// TIA Portal V19 export
FUNCTION_BLOCK "Convoyer7"   // FB6, F_LAD
{ S7_Optimized_Access := 'TRUE' }
   VAR_INPUT
      InverterStatus : "LDrvSafe_typeSinaTlg30Status";
      ESTOP : Bool;
      LIGHT_CURTAIN : Bool;
      PROCES_STAMPING : Bool;
      DOOR : Bool;
      FRQ_FEEDBACK : Bool;
      RESET : Bool;
   END_VAR
   VAR_OUTPUT
      InverterControl : "LDrvSafe_typeSinaTlg30Control";
      SAFETY_OK : Bool;
      INVERTER_OK : Bool;
      FRQ_NOK : Bool;
      REQ_RESET_ESTOP : Bool;
      SAFETY_VALVE : Bool;
   END_VAR
   VAR
      ESTOP_ON : Bool;
      INVERTER_FAULT : Bool;
      ESTOP1_Instance : ESTOP1;
      LDrvSafe_SinaTlg30Control_Instance : "LDrvSafe_SinaTlg30Control";
      LDrvSafe_SinaTlg30Status_Instance : "LDrvSafe_SinaTlg30Status";
   END_VAR
BEGIN

REGION Network 1
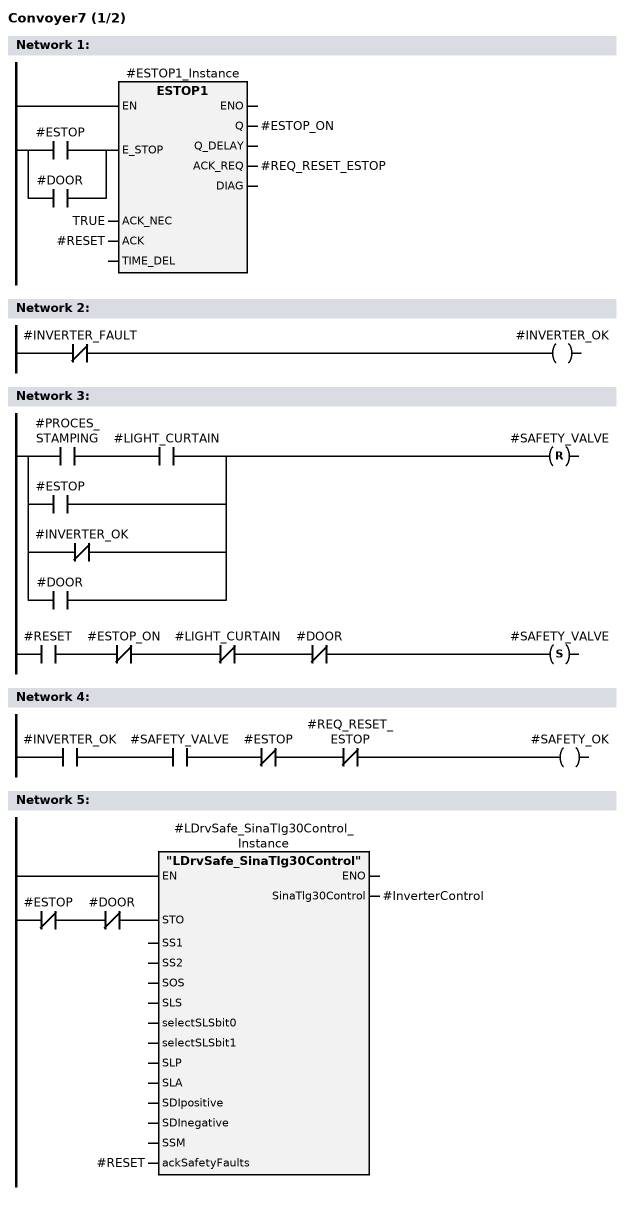
   RUNG wire#powerrail
      #ESTOP1_Instance.ESTOP1(E_STOP := wire#w1, ACK_NEC := TRUE, ACK := #RESET, TIME_DEL :=, Q => #ESTOP_ON, Q_DELAY =>, ACK_REQ => #REQ_RESET_ESTOP, DIAG =>)
   END_RUNG
   RUNG wire#powerrail
      Contact( #ESTOP )
   END_RUNG wire#w1
   RUNG wire#powerrail
      Contact( #DOOR )
   END_RUNG wire#w1
   // the same network as SCL:
   #ESTOP1_Instance(E_STOP := #ESTOP OR #DOOR,   // ESTOP1
                    ACK_NEC := TRUE,
                    ACK := #RESET,
                    Q => #ESTOP_ON,
                    ACK_REQ => #REQ_RESET_ESTOP);
END_REGION

REGION Network 2
   RUNG wire#powerrail
      I_Contact( #INVERTER_FAULT )
      Coil( #INVERTER_OK )
   END_RUNG
   // the same network as SCL:
   #INVERTER_OK := NOT #INVERTER_FAULT;
END_REGION

REGION Network 3
   RUNG wire#powerrail
      Contact( #PROCES_STAMPING )
      Contact( #LIGHT_CURTAIN )
      wire#w1
      R_Coil( #SAFETY_VALVE )
   END_RUNG
   RUNG wire#powerrail
      Contact( #ESTOP )
   END_RUNG wire#w1
   RUNG wire#powerrail
      I_Contact( #INVERTER_OK )
   END_RUNG wire#w1
   RUNG wire#powerrail
      Contact( #DOOR )
   END_RUNG wire#w1
   RUNG wire#powerrail
      Contact( #RESET )
      I_Contact( #ESTOP_ON )
      I_Contact( #LIGHT_CURTAIN )
      I_Contact( #DOOR )
      S_Coil( #SAFETY_VALVE )
   END_RUNG
   // the same network as SCL:
   IF (#PROCES_STAMPING AND #LIGHT_CURTAIN) OR #ESTOP OR NOT #INVERTER_OK OR #DOOR THEN
       #SAFETY_VALVE := FALSE;
   END_IF;
   IF #RESET AND NOT #ESTOP_ON AND NOT #LIGHT_CURTAIN AND NOT #DOOR THEN #SAFETY_VALVE := TRUE; END_IF;
END_REGION

REGION Network 4
   RUNG wire#powerrail
      Contact( #INVERTER_OK )
      Contact( #SAFETY_VALVE )
      I_Contact( #ESTOP )
      I_Contact( #REQ_RESET_ESTOP )
      Coil( #SAFETY_OK )
   END_RUNG
   // the same network as SCL:
   #SAFETY_OK := #INVERTER_OK AND #SAFETY_VALVE AND NOT #ESTOP AND NOT #REQ_RESET_ESTOP;
END_REGION

REGION Network 5
   RUNG wire#powerrail
      #LDrvSafe_SinaTlg30Control_Instance(STO := wire#w1, SS1 :=, SS2 :=, SOS :=, SLS :=, selectSLSbit0 :=, selectSLSbit1 :=, SLP :=, SLA :=, SDIpositive :=, SDInegative :=, SSM :=, ackSafetyFaults := #RESET, SinaTlg30Control => #InverterControl)
   END_RUNG
   RUNG wire#powerrail
      I_Contact( #ESTOP )
      I_Contact( #DOOR )
   END_RUNG wire#w1
   // the same network as SCL:
   #LDrvSafe_SinaTlg30Control_Instance(STO := NOT #ESTOP AND NOT #DOOR,   // "LDrvSafe_SinaTlg30Control"
                           ackSafetyFaults := #RESET,
                           SinaTlg30Control => #InverterControl);
END_REGION

REGION Network 6
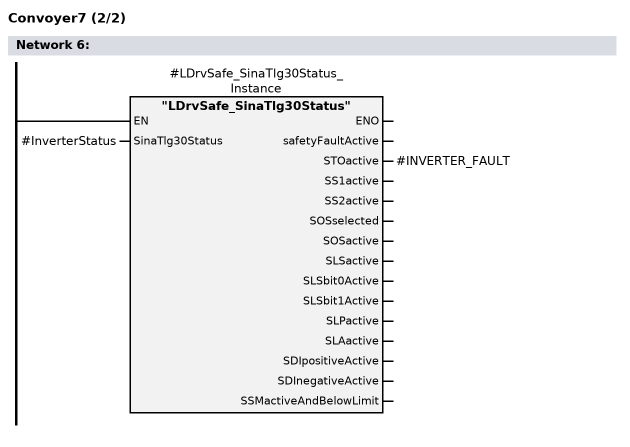
   RUNG wire#powerrail
      #LDrvSafe_SinaTlg30Status_Instance(SinaTlg30Status := #InverterStatus, safetyFaultActive =>, STOactive => #INVERTER_FAULT, SS1active =>, SS2active =>, SOSselected =>, SOSactive =>, SLSactive =>, SLSbit0Active =>, SLSbit1Active =>, SLPactive =>, SLAactive =>, SDIpositiveActive =>, SDInegativeActive =>, SSMactiveAndBelowLimit =>)
   END_RUNG
   // the same network as SCL:
   #LDrvSafe_SinaTlg30Status_Instance(SinaTlg30Status := #InverterStatus, STOactive => #INVERTER_FAULT);   // "LDrvSafe_SinaTlg30Status"
END_REGION
END_FUNCTION_BLOCK
